PROGRAM Fridge1
VAR
// Inputs (simulated)
	bDoorOpen : BOOL; // TRUE = door open
// Outputs
	bLight : BOOL; // Interior light
	nCounter : INT;
END_VAR
// Simple logic: light follows door state

bLight := bDoorOpen;
nCounter := nCounter + 1;

END_PROGRAM

(* stored: Version 1.1.0.1, ProductVersion 3.1.4026.18
   POU Fridge1: Id {a6eb933c-1bbb-440c-8cb2-d01941b2a718}, SpecialFunc None *)
